ABB RAPID module: test_right.mod

MODULE test_right
LOCAL CONST string YuMi_App_Program_Version:="1.0.1"; !Do not edit or remove this line!
LOCAL VAR robtarget s4 := [[289.792,-146.158,135.174],[0.280108,-0.240636,-0.733727,-0.570332],[0,-1,-3,10],[-100.003,9E+09,9E+09,9E+09,9E+09,9E+09]];
LOCAL VAR robtarget s3 := [[286.16,-168.529,202.758],[0.421955,-0.862656,0.0419983,-0.275708],[0,-2,-1,10],[-70.001,9E+09,9E+09,9E+09,9E+09,9E+09]];
LOCAL VAR robtarget s2 := [[289.814,-146.171,135.178],[0.28011,-0.240696,-0.733672,-0.570376],[0,-1,-2,10],[-99.9938,9E+09,9E+09,9E+09,9E+09,9E+09]];
LOCAL VAR robtarget s1 := [[286.157,-168.559,202.766],[0.421911,-0.862664,0.0420749,-0.275739],[0,-2,-1,10],[-69.9949,9E+09,9E+09,9E+09,9E+09,9E+09]];
PROC main()
MoveSync s1;
MoveSync s2;
MoveSync s3;
MoveSync s4;
ENDPROC
ENDMODULE
